TYPE ST_Axis :
STRUCT
	strName			:STRING					    ;
	wstrName		:WSTRING				    ;
	strNetID        :STRING;
	uiSlaveAddr     AT%I*  :WORD;
	Control			:ST_AxisControl				;		
	Parameter		:ST_AxisParameter			;		
	State			:ST_AxisState				;	
	Pos				:ST_AxisPos		            ;
END_STRUCT
END_TYPE

(* stored: Version 1.1.0.1, ProductVersion 3.1.4024.12
   DUT ST_Axis: Id {5caed6f4-603b-4f42-8951-9670a80a1dc7} *)
